FUNCTION_BLOCK FB_XmlPersistentEventStorage IMPLEMENTS I_PersistentEventStorage
VAR_INPUT
END_VAR
VAR_OUTPUT
END_VAR
VAR
END_VAR

{warning 'add method implementation '}
METHOD StoreEvent
VAR_INPUT
	stEvent	: ST_Event;
END_VAR
END_METHOD

END_FUNCTION_BLOCK

(* stored: Version 1.1.0.1, ProductVersion 3.1.4024.15
   POU FB_XmlPersistentEventStorage: Id {b6d466bf-6b6d-4c4d-a0a8-da7bfd6efc42}, SpecialFunc None
   Method StoreEvent: Id {44e4155d-7bf2-4577-b19d-81c1e94a07f5} *)
